(* Logix 5000 project; controller Thurs_Lab2 vendor 1 type 14 code 156 rev 30.11; software revision 30.00; part 2 of 5 *)
(* tags used below, declared in another part *)
   ALARM_CLOSE : BOOL;
   AUTO : BOOL;
   BLINK_PL1 : TIMER;
   BLINK_PL3 : TIMER;
   BLUE : BOOL;
   BLUE_BLINKER : TIMER;
   BLUE_STK : BOOL;
   BUTTON : BOOL;
   BYPASS : BOOL;
   CHECK_0 : BOOL;
   CHECK_1 : BOOL;
   CYCLE_START : BOOL;
   CYCLE_STOP : BOOL;
   CYL1_EXT_PX : BOOL;
   CYL1_RET_PX : BOOL;
   CYL2_EXT_4_LOAD_AND_UNLOAD : BOOL;
   CYL2_EXT_PX : BOOL;
   DEEP : COUNTER;
   DELAY_PE_INPUT_PSB : TIMER;
   DELAY_PE_INPUT_PSW : TIMER;
   DELAY_PE_INPUT_STATE : TIMER;
   DRILL2 : DRILL2;
   DRILL3 : DRILL3;
   DRILL4 : DRILL4;
   ESTOP : BOOL;
   ESTOP_PRESSED : BOOL;
   EXTEND : TIMER;
   FAILURE2LOAD : TIMER;
   FAILURE_2_LOAD : BOOL;
   FAULT : BOOL;
   FAULT_S : DINT;
   FAULTED : BOOL;
   FROM_CELL : FROM_CELL;
   GOOD_PART : BOOL;
   GREEN_BLINKER : TIMER;
   GREEN_STK : BOOL;
   INPUT : INT;
   LIMIT_PSB : BOOL;
   LIMIT_PSW : BOOL;
   LIMIT_STATE : BOOL;
   LOADING : BOOL;
   MACHINE_PAUSED : BOOL;
   Manual : BOOL;
   MARK_BLUE : BOOL;
   MARK_CYL1 : CYLINDER;
   MARK_GREEN : BOOL;
   MARK_LIGHTS : BOOL;
   MARK_RED : BOOL;
   MARK_WHITE_STK : BOOL;
   MARK_YELLOW : BOOL;
   MODE_SELECT : DINT;
   MOTOR_WHEEL_PE : BOOL;
   MSTER_RESET_TWCE : BOOL;
   ONESHOT1 : BOOL;
   ONESHOT2 : BOOL;
   ONESHOT3 : BOOL;
   OP1_STOP : BOOL;
   OP2_STEP : DINT;
   OP2_STOP : BOOL;
   OP2STEP : DINT;
   OP3_STOP : BOOL;
   OP4_STOP : BOOL;
   OP5_STATIC_OVER : BOOL;
   OP5_STATIC_UNDER : BOOL;
   OP5_STOP : BOOL;
   OP5_TEST : DINT;
   OP5_TEST_STATIC : DINT;
   OP6_OP7 : DINT;
   OP6_STOP : BOOL;
   OP7_STOP : BOOL;
   OPERATION : DINT;
   OPERATION_5_OVER : BOOL;
   OPERATION_5_REJECT : BOOL;
   OPERATION_5_UNDER : BOOL;
   OPERATION_7_OVER : BOOL;
   OPERATION_7_REJECT : BOOL;
   OPERATION_7_UNDER : BOOL;
   OPERATION_DONE : DINT;
   OPERATION_OFF : DINT;
   OUT_OF_INK_FAULT : BOOL;
   PART_NOT_PX : BOOL;
   PART_PX : BOOL;
   PAUSED : BOOL;
   PAUSED_OPERATION_1 : BOOL;
   PAUSED_OPERATION_5 : BOOL;
   PAUSED_OPERATION_7 : BOOL;
   PB0 : BOOL;
   PB1 : BOOL;
   PB2 : BOOL;
   PB3 : BOOL;
   PB4 : BOOL;
   PB5 : BOOL;
   PL1 : BOOL;
   PL3 : BOOL;
   PUSH : BOOL;
   PV_ANALOG_PROBE : DINT;
   PV_ANALOG_PROBE_STATIC : DINT;
   PV_CYL1_DEPTH : DINT;
   PV_CYL1_EXT_LIMIT : DINT;
   PV_CYL1_EXT_TIME : DINT;
   PV_DRILLING : DINT;
   PV_STOPPING : DINT;
   PV_UP2SPEED : DINT;
   RED_BLINKER : TIMER;
   RED_STK : BOOL;
   REJECT_FAULT : BOOL;
   RESET : BOOL;
   SAFETY_RELAY_OFF : BOOL;
   SEQ_EN : BOOL;
   SETTLE1 : TIMER;
   SHALLOW : COUNTER;
   SPARE : BOOL;
   STA : DINT;
   START_SIGNAL : BOOL;
   STATE : DINT;
   STATUS : DINT;
   STEP : DINT;
   Timer : TIMER;
   TIMER_1 : TIMER;
   TIMER_2 : TIMER;
   TO_CELL : TO_CELL;
   TOO_DEEP : BOOL;
   TOO_SHALLOW : BOOL;
   TRANSFER7 : TIMER;
   TRANSFER7_TIME_EXCEED : BOOL;
   TWO_HAND_START : BOOL;
   UNLOADING : BOOL;
   YELLOW_STK : BOOL;
(* MainProgram, continued *)

ROUTINE HMI_SCREEN   (* ladder *)
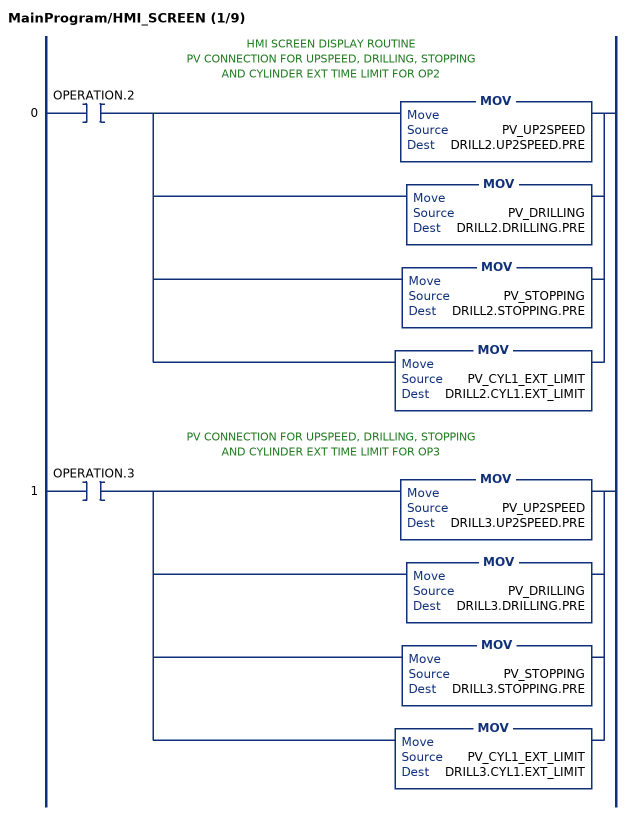
   // HMI SCREEN DISPLAY ROUTINE
   // PV CONNECTION FOR UPSPEED, DRILLING, STOPPING
   // AND CYLINDER EXT TIME LIMIT FOR OP2
   0: XIC(OPERATION.2)[MOV(PV_UP2SPEED,DRILL2.UP2SPEED.PRE) ,MOV(PV_DRILLING,DRILL2.DRILLING.PRE) ,MOV(PV_STOPPING,DRILL2.STOPPING.PRE) ,MOV(PV_CYL1_EXT_LIMIT,DRILL2.CYL1.EXT_LIMIT) ];
   // PV CONNECTION FOR UPSPEED, DRILLING, STOPPING
   // AND CYLINDER EXT TIME LIMIT FOR OP3
   1: XIC(OPERATION.3)[MOV(PV_UP2SPEED,DRILL3.UP2SPEED.PRE) ,MOV(PV_DRILLING,DRILL3.DRILLING.PRE) ,MOV(PV_STOPPING,DRILL3.STOPPING.PRE) ,MOV(PV_CYL1_EXT_LIMIT,DRILL3.CYL1.EXT_LIMIT) ];
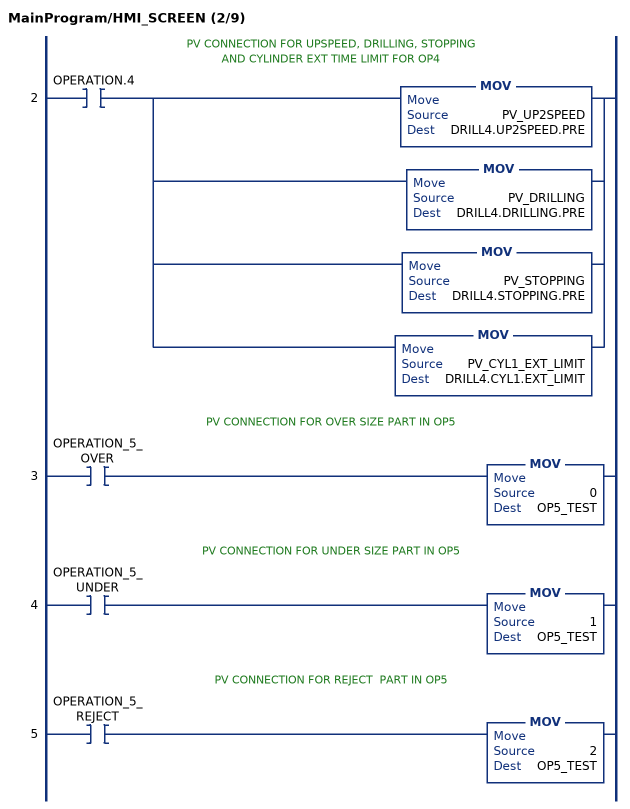
   // PV CONNECTION FOR UPSPEED, DRILLING, STOPPING
   // AND CYLINDER EXT TIME LIMIT FOR OP4
   2: XIC(OPERATION.4)[MOV(PV_UP2SPEED,DRILL4.UP2SPEED.PRE) ,MOV(PV_DRILLING,DRILL4.DRILLING.PRE) ,MOV(PV_STOPPING,DRILL4.STOPPING.PRE) ,MOV(PV_CYL1_EXT_LIMIT,DRILL4.CYL1.EXT_LIMIT) ];
   // PV CONNECTION FOR OVER SIZE PART IN OP5
   3: XIC(OPERATION_5_OVER)MOV(0,OP5_TEST);
   // PV CONNECTION FOR UNDER SIZE PART IN OP5
   4: XIC(OPERATION_5_UNDER)MOV(1,OP5_TEST);
   // PV CONNECTION FOR REJECT  PART IN OP5
   5: XIC(OPERATION_5_REJECT)MOV(2,OP5_TEST);
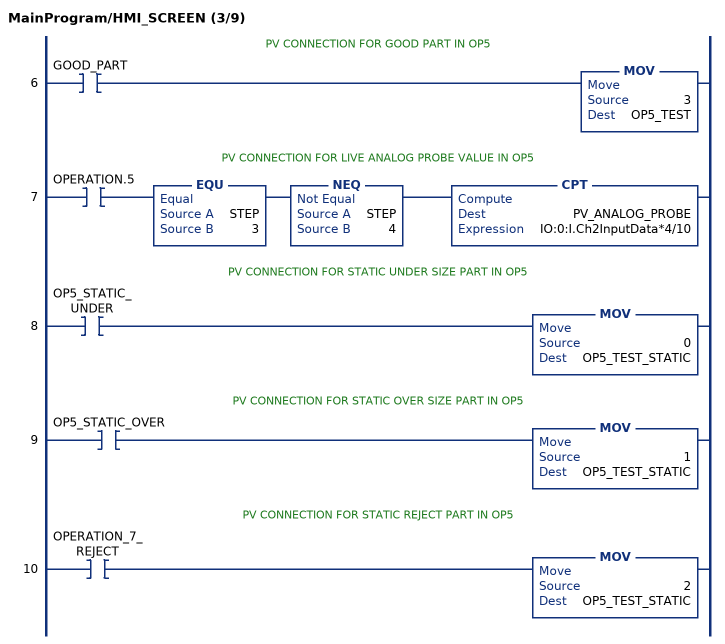
   // PV CONNECTION FOR GOOD PART IN OP5
   6: XIC(GOOD_PART)MOV(3,OP5_TEST);
   // PV CONNECTION FOR LIVE ANALOG PROBE VALUE IN OP5
   7: XIC(OPERATION.5)EQU(STEP,3)NEQ(STEP,4)CPT(PV_ANALOG_PROBE,IO:0:I.Ch2InputData*4/10);
   // PV CONNECTION FOR STATIC UNDER SIZE PART IN OP5
   8: XIC(OP5_STATIC_UNDER)MOV(0,OP5_TEST_STATIC);
   // PV CONNECTION FOR STATIC OVER SIZE PART IN OP5
   9: XIC(OP5_STATIC_OVER)MOV(1,OP5_TEST_STATIC);
   // PV CONNECTION FOR STATIC REJECT PART IN OP5
   10: XIC(OPERATION_7_REJECT)MOV(2,OP5_TEST_STATIC);
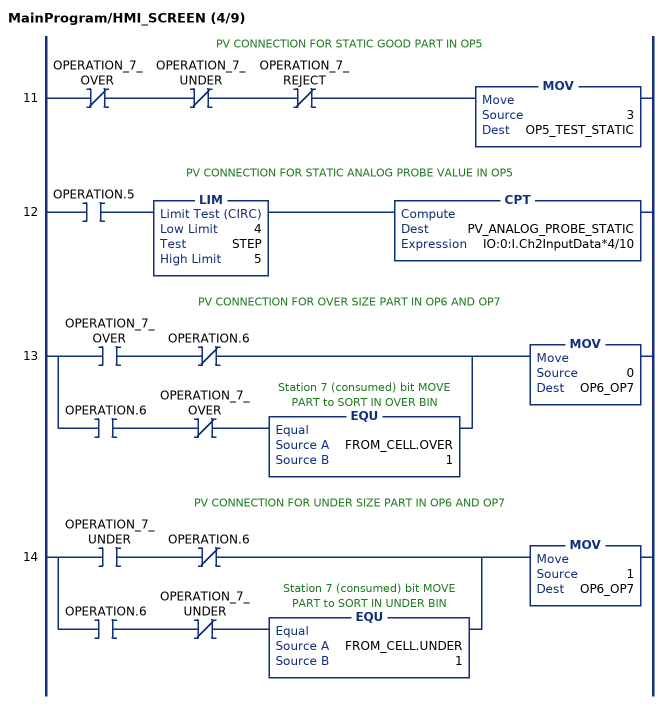
   // PV CONNECTION FOR STATIC GOOD PART IN OP5
   11: XIO(OPERATION_7_OVER)XIO(OPERATION_7_UNDER)XIO(OPERATION_7_REJECT)MOV(3,OP5_TEST_STATIC);
   // PV CONNECTION FOR STATIC ANALOG PROBE VALUE IN OP5
   12: XIC(OPERATION.5)LIM(4,STEP,5)CPT(PV_ANALOG_PROBE_STATIC,IO:0:I.Ch2InputData*4/10);
   // PV CONNECTION FOR OVER SIZE PART IN OP6 AND OP7
   13: [XIC(OPERATION_7_OVER) XIO(OPERATION.6) ,XIC(OPERATION.6) XIO(OPERATION_7_OVER) EQU(FROM_CELL.OVER,1) ]MOV(0,OP6_OP7);
   // PV CONNECTION FOR UNDER SIZE PART IN OP6 AND OP7
   14: [XIC(OPERATION_7_UNDER) XIO(OPERATION.6) ,XIC(OPERATION.6) XIO(OPERATION_7_UNDER) EQU(FROM_CELL.UNDER,1) ]MOV(1,OP6_OP7);
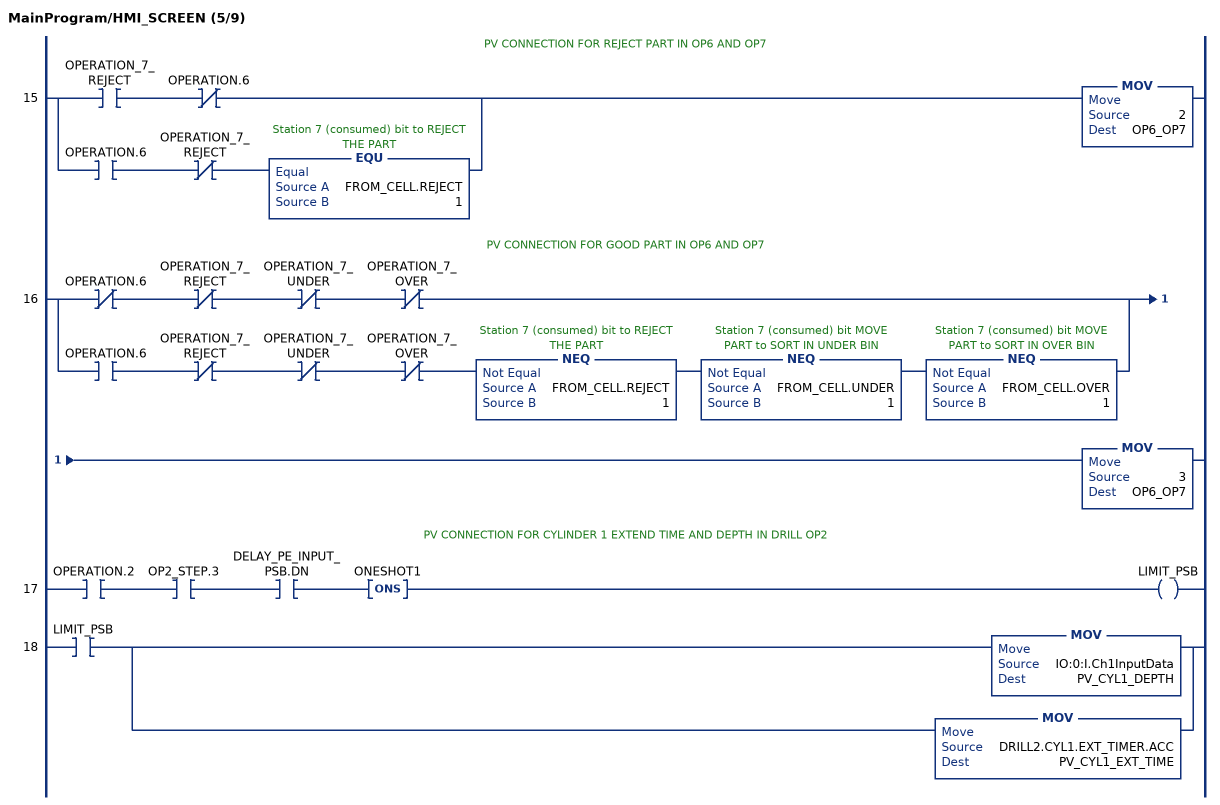
   // PV CONNECTION FOR REJECT PART IN OP6 AND OP7
   15: [XIC(OPERATION_7_REJECT) XIO(OPERATION.6) ,XIC(OPERATION.6) XIO(OPERATION_7_REJECT) EQU(FROM_CELL.REJECT,1) ]MOV(2,OP6_OP7);
   // PV CONNECTION FOR GOOD PART IN OP6 AND OP7
   16: [XIO(OPERATION.6) XIO(OPERATION_7_REJECT) XIO(OPERATION_7_UNDER) XIO(OPERATION_7_OVER) ,XIC(OPERATION.6) XIO(OPERATION_7_REJECT) XIO(OPERATION_7_UNDER) XIO(OPERATION_7_OVER) NEQ(FROM_CELL.REJECT,1) NEQ(FROM_CELL.UNDER,1) NEQ(FROM_CELL.OVER,1) ]MOV(3,OP6_OP7);
   // PV CONNECTION FOR CYLINDER 1 EXTEND TIME AND DEPTH IN DRILL OP2
   17: XIC(OPERATION.2)XIC(OP2_STEP.3)XIC(DELAY_PE_INPUT_PSB.DN)ONS(ONESHOT1)OTE(LIMIT_PSB);
   18: XIC(LIMIT_PSB)[MOV(IO:0:I.Ch1InputData,PV_CYL1_DEPTH) ,MOV(DRILL2.CYL1.EXT_TIMER.ACC,PV_CYL1_EXT_TIME) ];
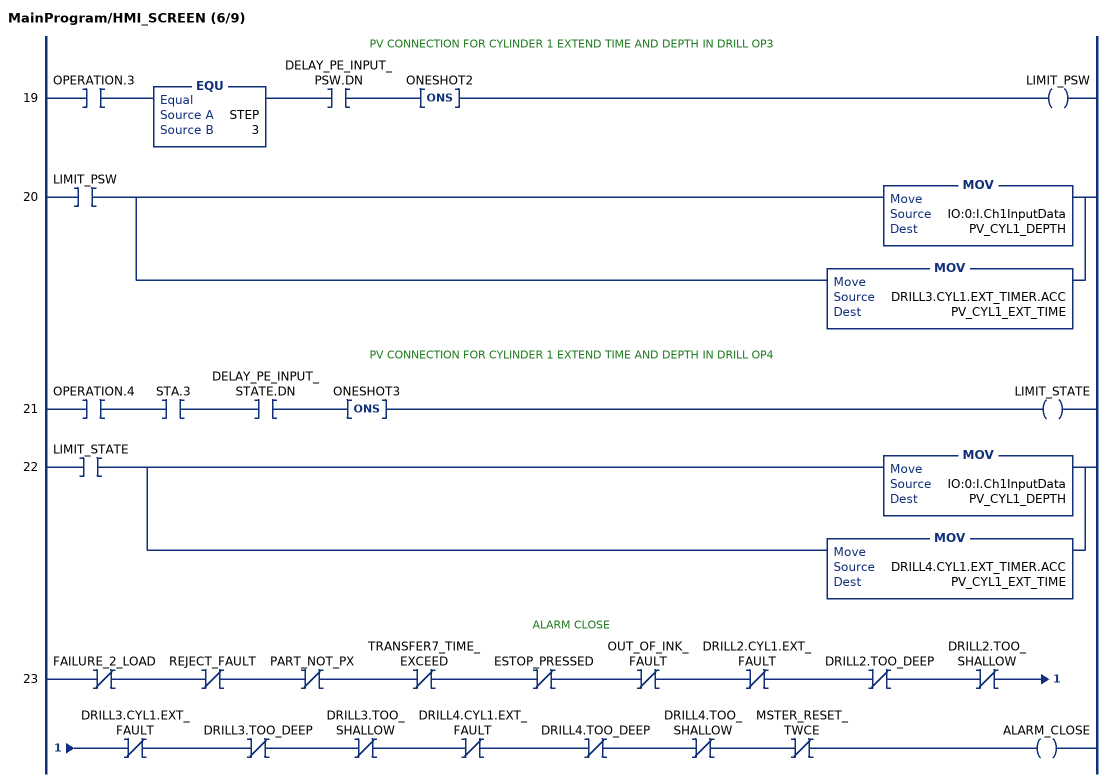
   // PV CONNECTION FOR CYLINDER 1 EXTEND TIME AND DEPTH IN DRILL OP3
   19: XIC(OPERATION.3)EQU(STEP,3)XIC(DELAY_PE_INPUT_PSW.DN)ONS(ONESHOT2)OTE(LIMIT_PSW);
   20: XIC(LIMIT_PSW)[MOV(IO:0:I.Ch1InputData,PV_CYL1_DEPTH) ,MOV(DRILL3.CYL1.EXT_TIMER.ACC,PV_CYL1_EXT_TIME) ];
   // PV CONNECTION FOR CYLINDER 1 EXTEND TIME AND DEPTH IN DRILL OP4
   21: XIC(OPERATION.4)XIC(STA.3)XIC(DELAY_PE_INPUT_STATE.DN)ONS(ONESHOT3)OTE(LIMIT_STATE);
   22: XIC(LIMIT_STATE)[MOV(IO:0:I.Ch1InputData,PV_CYL1_DEPTH) ,MOV(DRILL4.CYL1.EXT_TIMER.ACC,PV_CYL1_EXT_TIME) ];
   // ALARM CLOSE
   23: XIO(FAILURE_2_LOAD)XIO(REJECT_FAULT)XIO(PART_NOT_PX)XIO(TRANSFER7_TIME_EXCEED)XIO(ESTOP_PRESSED)XIO(OUT_OF_INK_FAULT)XIO(DRILL2.CYL1.EXT_FAULT)XIO(DRILL2.TOO_DEEP)XIO(DRILL2.TOO_SHALLOW)XIO(DRILL3.CYL1.EXT_FAULT)XIO(DRILL3.TOO_DEEP)XIO(DRILL3.TOO_SHALLOW)XIO(DRILL4.CYL1.EXT_FAULT)XIO(DRILL4.TOO_DEEP)XIO(DRILL4.TOO_SHALLOW)XIO(MSTER_RESET_TWCE)OTE(ALARM_CLOSE);
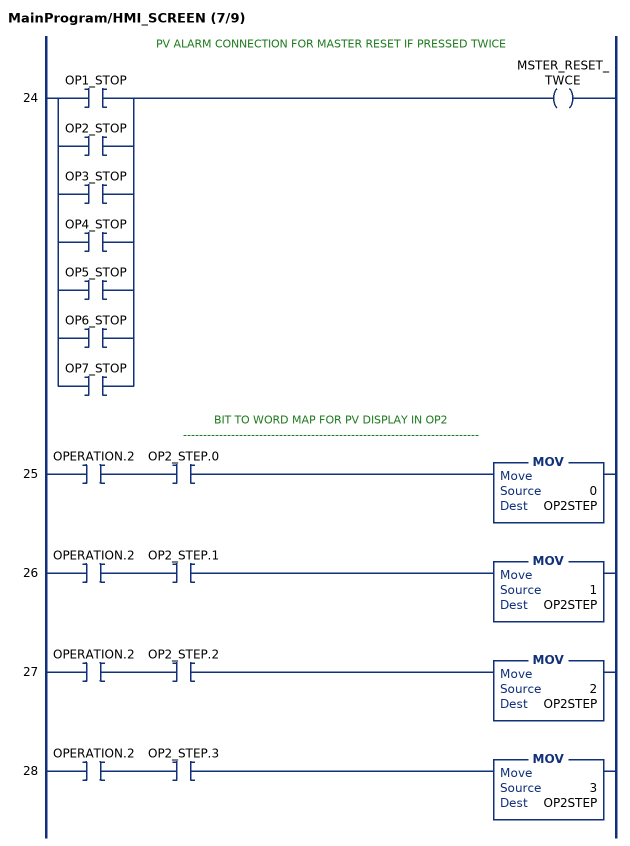
   // PV ALARM CONNECTION FOR MASTER RESET IF PRESSED TWICE
   24: [XIC(OP1_STOP) ,XIC(OP2_STOP) ,XIC(OP3_STOP) ,XIC(OP4_STOP) ,XIC(OP5_STOP) ,XIC(OP6_STOP) ,XIC(OP7_STOP) ]OTE(MSTER_RESET_TWCE);
   // BIT TO WORD MAP FOR PV DISPLAY IN OP2
   // --------------------------------------------------------------------------
   25: XIC(OPERATION.2)XIC(OP2_STEP.0)MOV(0,OP2STEP);
   26: XIC(OPERATION.2)XIC(OP2_STEP.1)MOV(1,OP2STEP);
   27: XIC(OPERATION.2)XIC(OP2_STEP.2)MOV(2,OP2STEP);
   28: XIC(OPERATION.2)XIC(OP2_STEP.3)MOV(3,OP2STEP);
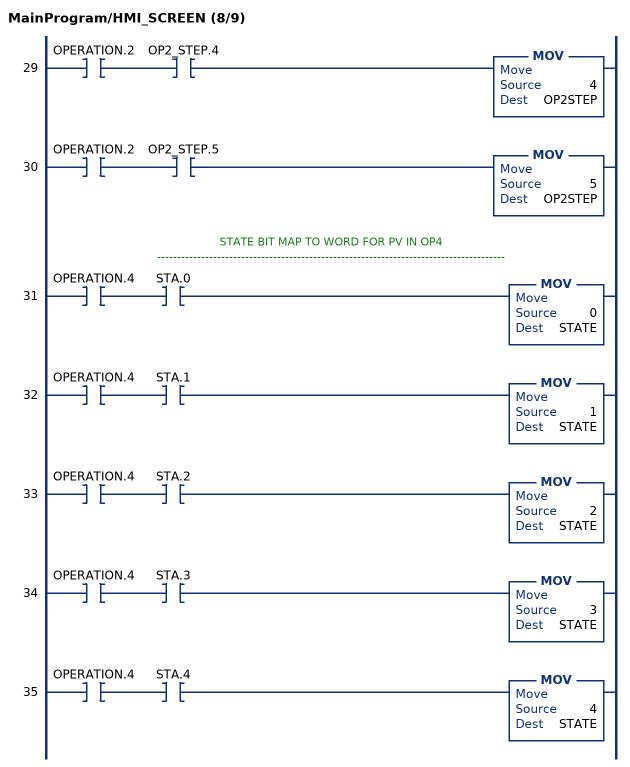
   29: XIC(OPERATION.2)XIC(OP2_STEP.4)MOV(4,OP2STEP);
   30: XIC(OPERATION.2)XIC(OP2_STEP.5)MOV(5,OP2STEP);
   // STATE BIT MAP TO WORD FOR PV IN OP4
   // ---------------------------------------------------------------------------------------
   31: XIC(OPERATION.4)XIC(STA.0)MOV(0,STATE);
   32: XIC(OPERATION.4)XIC(STA.1)MOV(1,STATE);
   33: XIC(OPERATION.4)XIC(STA.2)MOV(2,STATE);
   34: XIC(OPERATION.4)XIC(STA.3)MOV(3,STATE);
   35: XIC(OPERATION.4)XIC(STA.4)MOV(4,STATE);
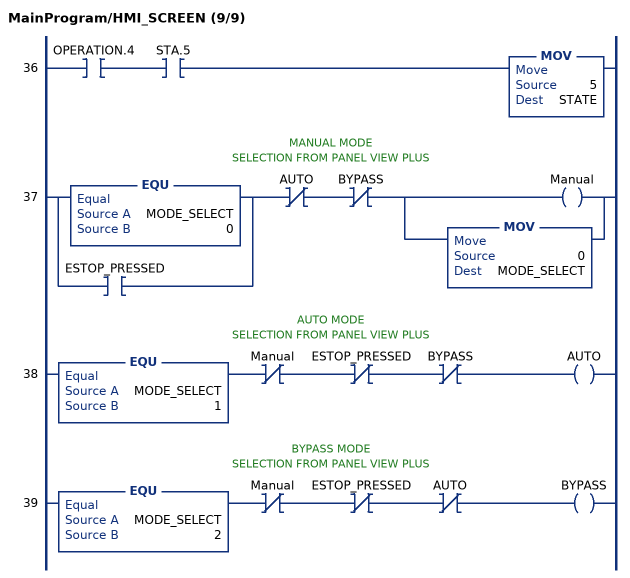
   36: XIC(OPERATION.4)XIC(STA.5)MOV(5,STATE);
   // MANUAL MODE
   // SELECTION FROM PANEL VIEW PLUS
   37: [EQU(MODE_SELECT,0) ,XIC(ESTOP_PRESSED) ]XIO(AUTO)XIO(BYPASS)[OTE(Manual) ,MOV(0,MODE_SELECT) ];
   // AUTO MODE
   // SELECTION FROM PANEL VIEW PLUS
   38: EQU(MODE_SELECT,1)XIO(Manual)XIO(ESTOP_PRESSED)XIO(BYPASS)OTE(AUTO);
   // BYPASS MODE
   // SELECTION FROM PANEL VIEW PLUS
   39: EQU(MODE_SELECT,2)XIO(Manual)XIO(ESTOP_PRESSED)XIO(AUTO)OTE(BYPASS);
END_ROUTINE

ROUTINE INDICATOR   (* ladder *)
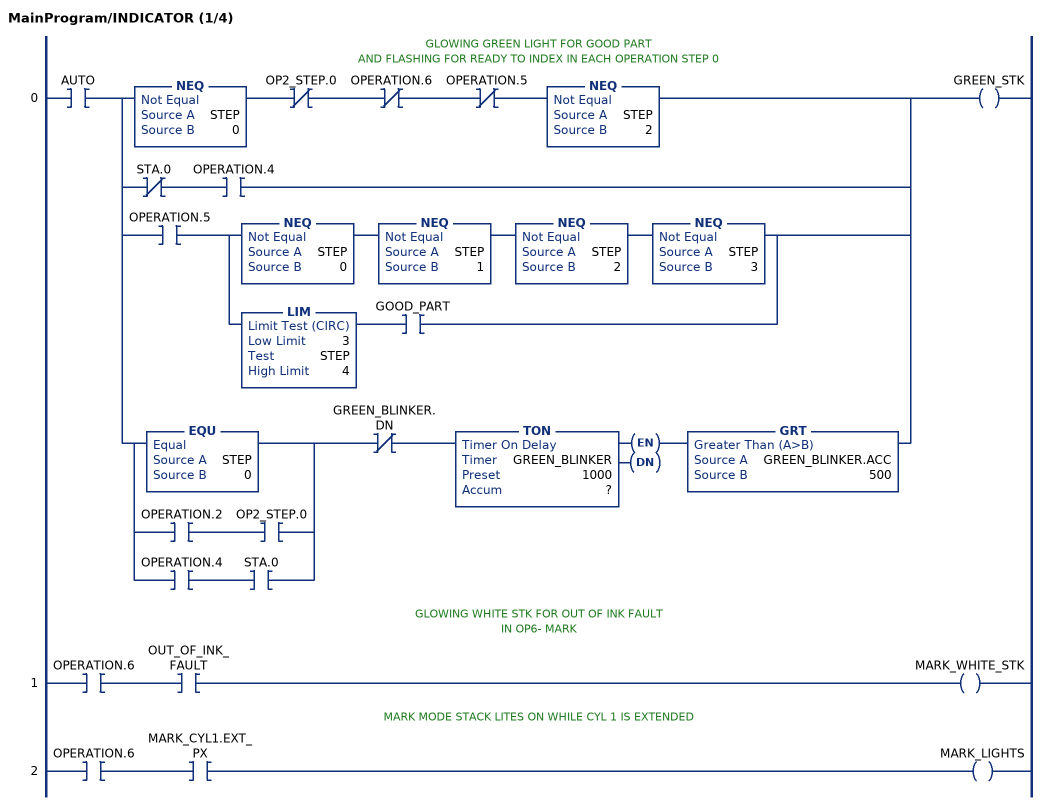
   // GLOWING GREEN LIGHT FOR GOOD PART
   // AND FLASHING FOR READY TO INDEX IN EACH OPERATION STEP 0
   0: XIC(AUTO)[[[NEQ(STEP,0) XIO(OP2_STEP.0) XIO(OPERATION.6) XIO(OPERATION.5) NEQ(STEP,2) ,XIO(STA.0) XIC(OPERATION.4) ] ,XIC(OPERATION.5) [NEQ(STEP,0) NEQ(STEP,1) NEQ(STEP,2) NEQ(STEP,3) ,LIM(3,STEP,4) XIC(GOOD_PART) ] ] ,[EQU(STEP,0) ,XIC(OPERATION.2) XIC(OP2_STEP.0) ,XIC(OPERATION.4) XIC(STA.0) ] XIO(GREEN_BLINKER.DN) TON(GREEN_BLINKER,?,?) GRT(GREEN_BLINKER.ACC,500) ]OTE(GREEN_STK);
   // GLOWING WHITE STK FOR OUT OF INK FAULT
   // IN OP6- MARK
   1: XIC(OPERATION.6)XIC(OUT_OF_INK_FAULT)OTE(MARK_WHITE_STK);
   // MARK MODE STACK LITES ON WHILE CYL 1 IS EXTENDED
   2: XIC(OPERATION.6)XIC(MARK_CYL1.EXT_PX)OTE(MARK_LIGHTS);
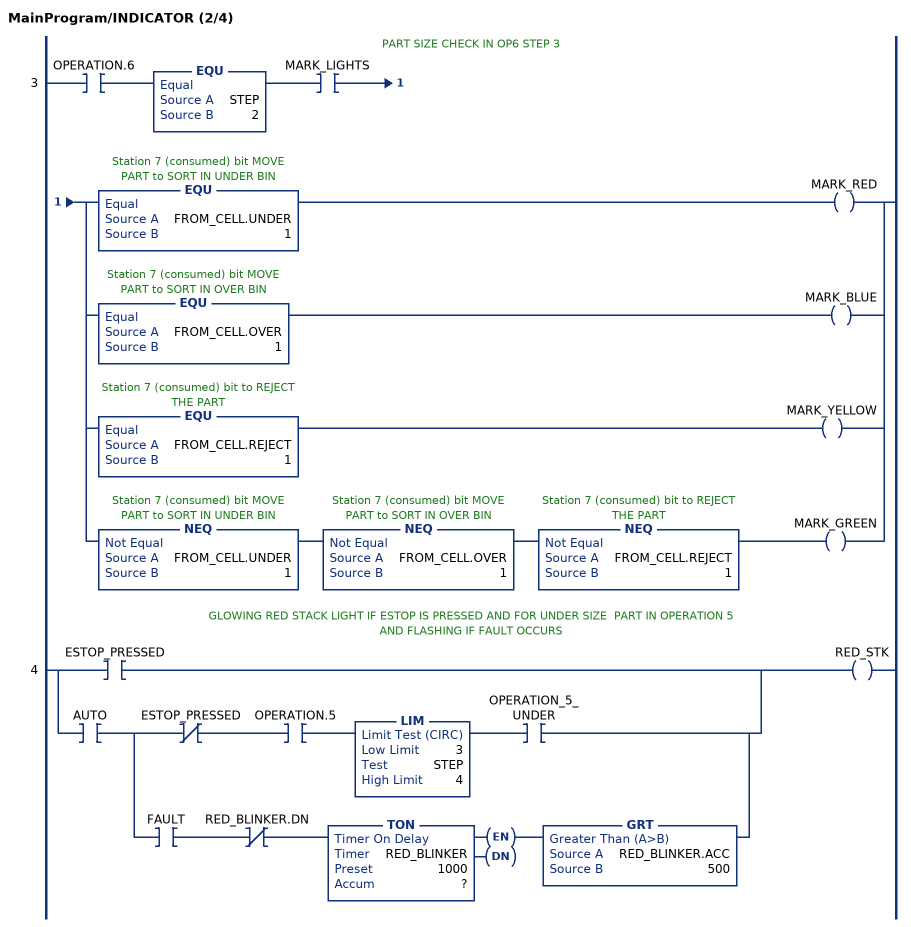
   // PART SIZE CHECK IN OP6 STEP 3
   3: XIC(OPERATION.6)EQU(STEP,2)XIC(MARK_LIGHTS)[EQU(FROM_CELL.UNDER,1) OTE(MARK_RED) ,EQU(FROM_CELL.OVER,1) OTE(MARK_BLUE) ,EQU(FROM_CELL.REJECT,1) OTE(MARK_YELLOW) ,NEQ(FROM_CELL.UNDER,1) NEQ(FROM_CELL.OVER,1) NEQ(FROM_CELL.REJECT,1) OTE(MARK_GREEN) ];
   // GLOWING RED STACK LIGHT IF ESTOP IS PRESSED AND FOR UNDER SIZE  PART IN OPERATION 5
   // AND FLASHING IF FAULT OCCURS
   4: [XIC(ESTOP_PRESSED) ,XIC(AUTO) [XIO(ESTOP_PRESSED) XIC(OPERATION.5) LIM(3,STEP,4) XIC(OPERATION_5_UNDER) ,XIC(FAULT) XIO(RED_BLINKER.DN) TON(RED_BLINKER,?,?) GRT(RED_BLINKER.ACC,500) ] ]OTE(RED_STK);
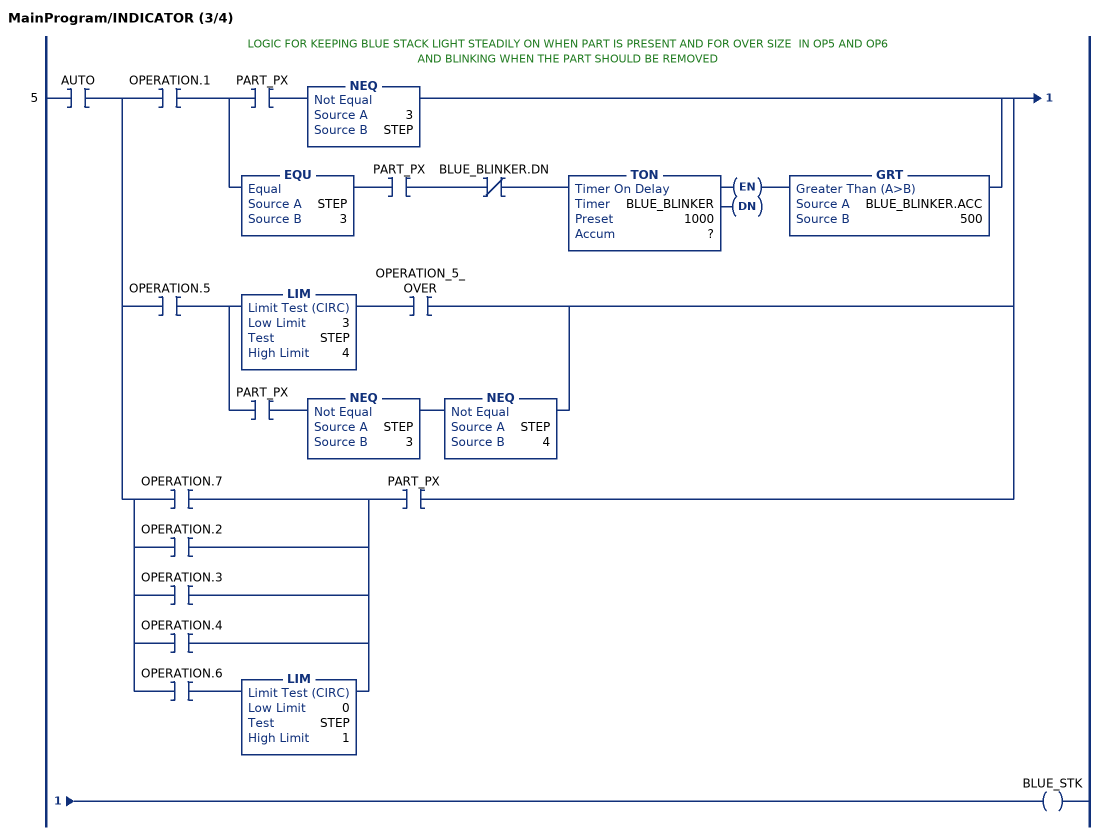
   // LOGIC FOR KEEPING BLUE STACK LIGHT STEADILY ON WHEN PART IS PRESENT AND FOR OVER SIZE  IN OP5 AND OP6
   // AND BLINKING WHEN THE PART SHOULD BE REMOVED
   5: XIC(AUTO)[XIC(OPERATION.1) [XIC(PART_PX) NEQ(3,STEP) ,EQU(STEP,3) XIC(PART_PX) XIO(BLUE_BLINKER.DN) TON(BLUE_BLINKER,?,?) GRT(BLUE_BLINKER.ACC,500) ] ,XIC(OPERATION.5) [LIM(3,STEP,4) XIC(OPERATION_5_OVER) ,XIC(PART_PX) NEQ(STEP,3) NEQ(STEP,4) ] ,[XIC(OPERATION.7) ,XIC(OPERATION.2) ,XIC(OPERATION.3) ,XIC(OPERATION.4) ,XIC(OPERATION.6) LIM(0,STEP,1) ] XIC(PART_PX) ]OTE(BLUE_STK);
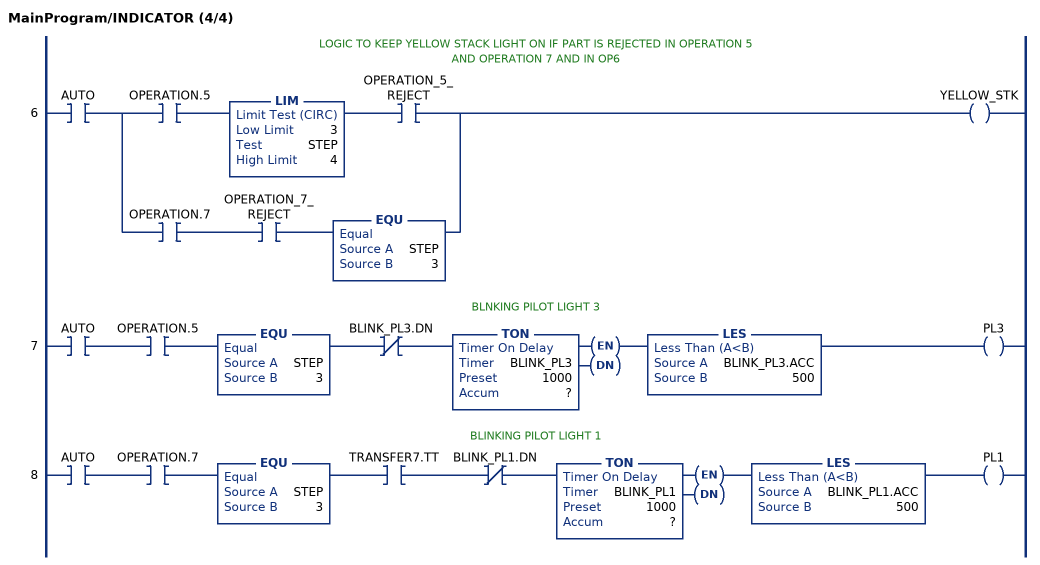
   // LOGIC TO KEEP YELLOW STACK LIGHT ON IF PART IS REJECTED IN OPERATION 5
   // AND OPERATION 7 AND IN OP6
   6: XIC(AUTO)[XIC(OPERATION.5) LIM(3,STEP,4) XIC(OPERATION_5_REJECT) ,XIC(OPERATION.7) XIC(OPERATION_7_REJECT) EQU(STEP,3) ]OTE(YELLOW_STK);
   // BLNKING PILOT LIGHT 3
   7: XIC(AUTO)XIC(OPERATION.5)EQU(STEP,3)XIO(BLINK_PL3.DN)TON(BLINK_PL3,?,?)LES(BLINK_PL3.ACC,500)OTE(PL3);
   // BLINKING PILOT LIGHT 1
   8: XIC(AUTO)XIC(OPERATION.7)EQU(STEP,3)XIC(TRANSFER7.TT)XIO(BLINK_PL1.DN)TON(BLINK_PL1,?,?)LES(BLINK_PL1.ACC,500)OTE(PL1);
END_ROUTINE

ROUTINE INPUT_BUFFERING   (* structured text *)
   // STRUCTURED TEXT PROGRAMMING FOR INPUT BUFFERING ROUTINE
   
   PB0 := Local:1:I.Data.0; // BUFFERING FOR PUSH BUTTON 0
   PB1 := Local:1:I.Data.1; //	BUFFERING FOR PUSH BUTTON 1
   PB2 := Local:1:I.Data.2; //	BUFFERING FOR PUSH BUTTON 2
   PB3 := Local:1:I.Data.3; //	BUFFERING FOR PUSH BUTTON 3
   PB4 := Local:1:I.Data.4; //	BUFFERING FOR PUSH BUTTON 4
   PB5 := Local:1:I.Data.5; //	BUFFERING FOR PUSH BUTTON 5
   
   CYL2_EXT_PX := Local:1:I.Data.6; //	BUFFERING FOR CYLINDER 2 EXTEND PROX
   MOTOR_WHEEL_PE:= Local:1:I.Data.7;	//	BUFFERING FOR MOTOR WHEEL PHOTO EYE
   PART_PX := Local:1:I.Data.8 AND (NOT PB2); //	BUFFERING FOR PART PRESENT AND INTERLOCKED WITH PB2
   SPARE:= Local:1:I.Data.9;
   
   CYL1_EXT_PX := Local:1:I.Data.10; //	BUFFERING CYLINDER 1 EXT PROX
   DRILL2.CYL1.EXT_PX := Local:1:I.Data.10;
   DRILL3.CYL1.EXT_PX := Local:1:I.Data.10;
   DRILL4.CYL1.EXT_PX := Local:1:I.Data.10;
   MARK_CYL1.EXT_PX := Local:1:I.Data.10;
   
   CYL1_RET_PX := Local:1:I.Data.11; //	BUFFERING FOR CYLINDER 1 EXTEND PROX
   DRILL2.CYL1.RET_PX := Local:1:I.Data.11;
   DRILL3.CYL1.RET_PX:= Local:1:I.Data.11;
   DRILL4.CYL1.RET_PX := Local:1:I.Data.11;
   MARK_CYL1.RET_PX := Local:1:I.Data.11;
   
   CYCLE_STOP := Local:1:I.Data.12;	//	BUFFERING FOR CYCLE STOP
   CYCLE_START := Local:1:I.Data.13;	//	BUFFERING FOR CYCLE START
   ESTOP_PRESSED := Local:1:I.Data.14;  //	BUFFERING FOR ESTOP PRESS
   SAFETY_RELAY_OFF:= Local:1:I.Data.15; // BUFFERING FOR SAFETY RELAY
   
   
   
END_ROUTINE

ROUTINE LOAD_UNLOADING   (* ladder *)
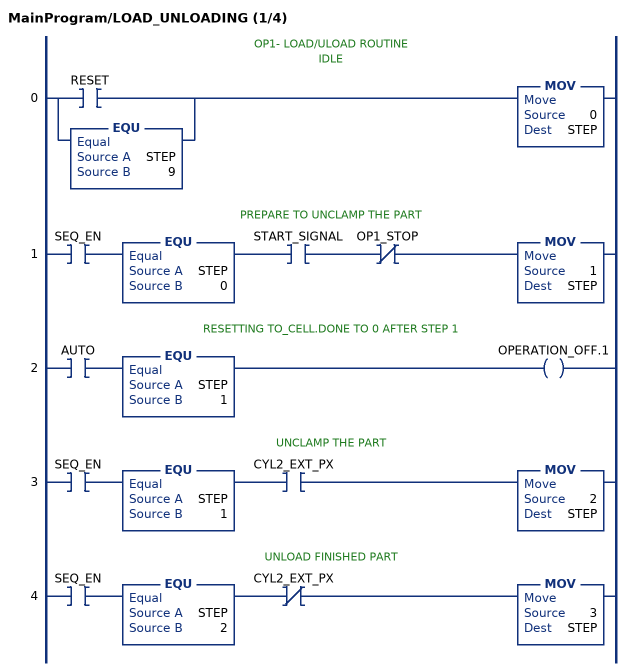
   // OP1- LOAD/ULOAD ROUTINE
   // IDLE
   0: [XIC(RESET) ,EQU(STEP,9) ]MOV(0,STEP);
   // PREPARE TO UNCLAMP THE PART
   1: XIC(SEQ_EN)EQU(STEP,0)XIC(START_SIGNAL)XIO(OP1_STOP)MOV(1,STEP);
   // RESETTING TO_CELL.DONE TO 0 AFTER STEP 1
   2: XIC(AUTO)EQU(STEP,1)OTE(OPERATION_OFF.1);
   // UNCLAMP THE PART
   3: XIC(SEQ_EN)EQU(STEP,1)XIC(CYL2_EXT_PX)MOV(2,STEP);
   // UNLOAD FINISHED PART
   4: XIC(SEQ_EN)EQU(STEP,2)XIO(CYL2_EXT_PX)MOV(3,STEP);
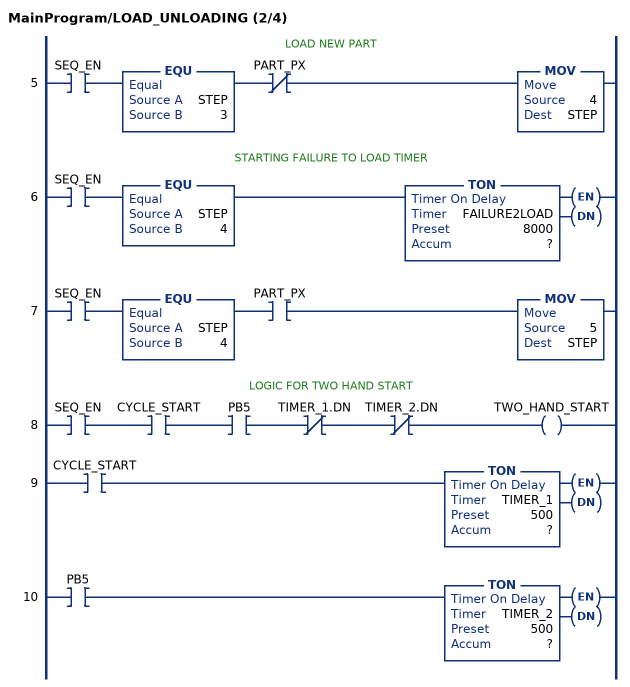
   // LOAD NEW PART
   5: XIC(SEQ_EN)EQU(STEP,3)XIO(PART_PX)MOV(4,STEP);
   // STARTING FAILURE TO LOAD TIMER
   6: XIC(SEQ_EN)EQU(STEP,4)TON(FAILURE2LOAD,?,?);
   7: XIC(SEQ_EN)EQU(STEP,4)XIC(PART_PX)MOV(5,STEP);
   // LOGIC FOR TWO HAND START
   8: XIC(SEQ_EN)XIC(CYCLE_START)XIC(PB5)XIO(TIMER_1.DN)XIO(TIMER_2.DN)OTE(TWO_HAND_START);
   9: XIC(CYCLE_START)TON(TIMER_1,?,?);
   10: XIC(PB5)TON(TIMER_2,?,?);
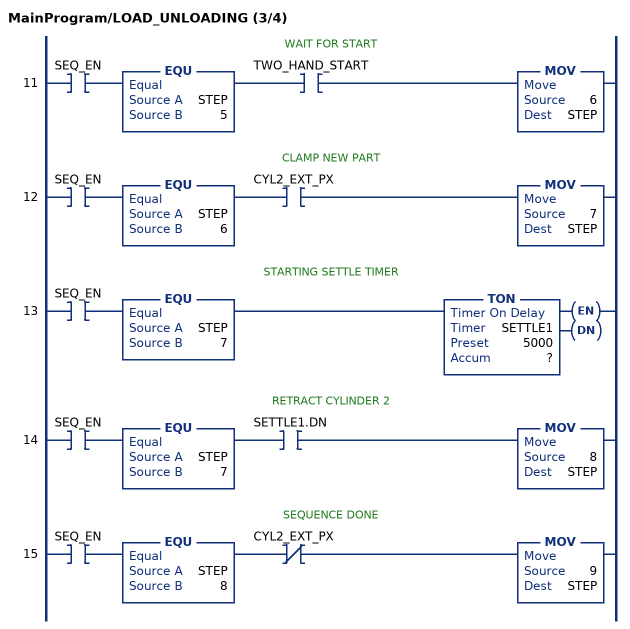
   // WAIT FOR START
   11: XIC(SEQ_EN)EQU(STEP,5)XIC(TWO_HAND_START)MOV(6,STEP);
   // CLAMP NEW PART
   12: XIC(SEQ_EN)EQU(STEP,6)XIC(CYL2_EXT_PX)MOV(7,STEP);
   // STARTING SETTLE TIMER
   13: XIC(SEQ_EN)EQU(STEP,7)TON(SETTLE1,?,?);
   // RETRACT CYLINDER 2
   14: XIC(SEQ_EN)EQU(STEP,7)XIC(SETTLE1.DN)MOV(8,STEP);
   // SEQUENCE DONE
   15: XIC(SEQ_EN)EQU(STEP,8)XIO(CYL2_EXT_PX)MOV(9,STEP);
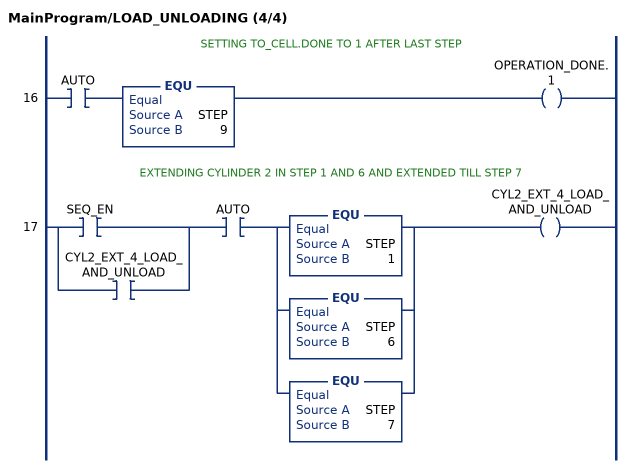
   // SETTING TO_CELL.DONE TO 1 AFTER LAST STEP
   16: XIC(AUTO)EQU(STEP,9)OTE(OPERATION_DONE.1);
   // EXTENDING CYLINDER 2 IN STEP 1 AND 6 AND EXTENDED TILL STEP 7
   17: [XIC(SEQ_EN) ,XIC(CYL2_EXT_4_LOAD_AND_UNLOAD) ]XIC(AUTO)[EQU(STEP,1) ,EQU(STEP,6) ,EQU(STEP,7) ]OTE(CYL2_EXT_4_LOAD_AND_UNLOAD);
END_ROUTINE

ROUTINE MACHINE_STATUS_AND_FAULTS   (* ladder *)
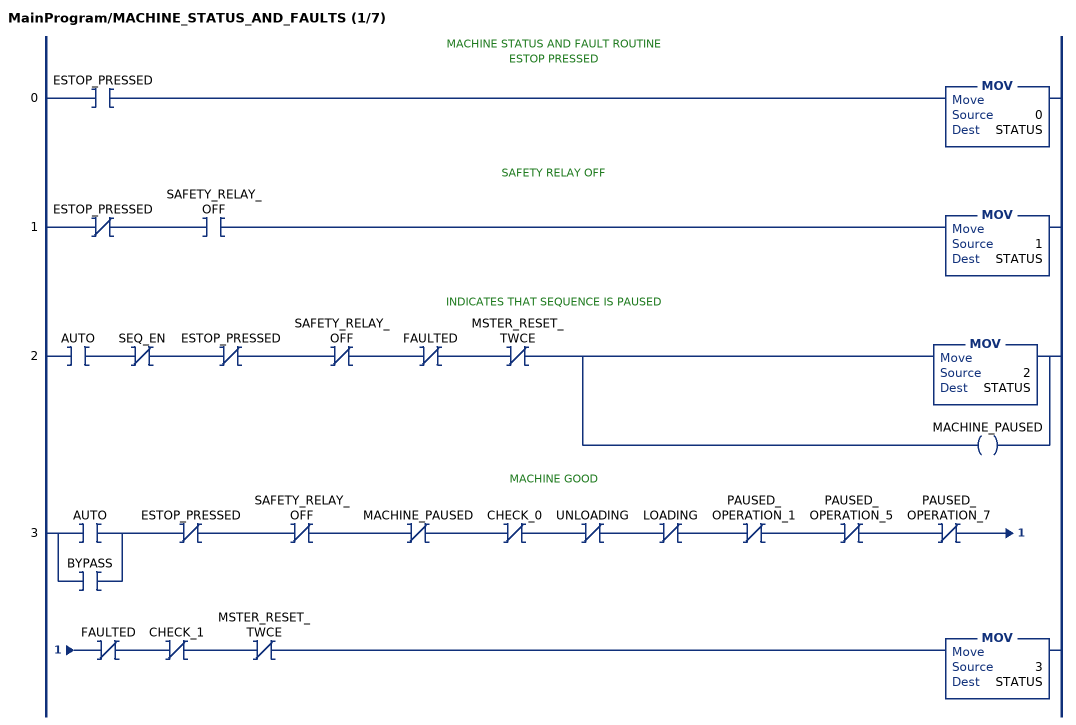
   // MACHINE STATUS AND FAULT ROUTINE
   // ESTOP PRESSED
   0: XIC(ESTOP_PRESSED)MOV(0,STATUS);
   // SAFETY RELAY OFF
   1: XIO(ESTOP_PRESSED)XIC(SAFETY_RELAY_OFF)MOV(1,STATUS);
   // INDICATES THAT SEQUENCE IS PAUSED
   2: XIC(AUTO)XIO(SEQ_EN)XIO(ESTOP_PRESSED)XIO(SAFETY_RELAY_OFF)XIO(FAULTED)XIO(MSTER_RESET_TWCE)[MOV(2,STATUS) ,OTE(MACHINE_PAUSED) ];
   // MACHINE GOOD
   3: [XIC(AUTO) ,XIC(BYPASS) ]XIO(ESTOP_PRESSED)XIO(SAFETY_RELAY_OFF)XIO(MACHINE_PAUSED)XIO(CHECK_0)XIO(UNLOADING)XIO(LOADING)XIO(PAUSED_OPERATION_1)XIO(PAUSED_OPERATION_5)XIO(PAUSED_OPERATION_7)XIO(FAULTED)XIO(CHECK_1)XIO(MSTER_RESET_TWCE)MOV(3,STATUS);
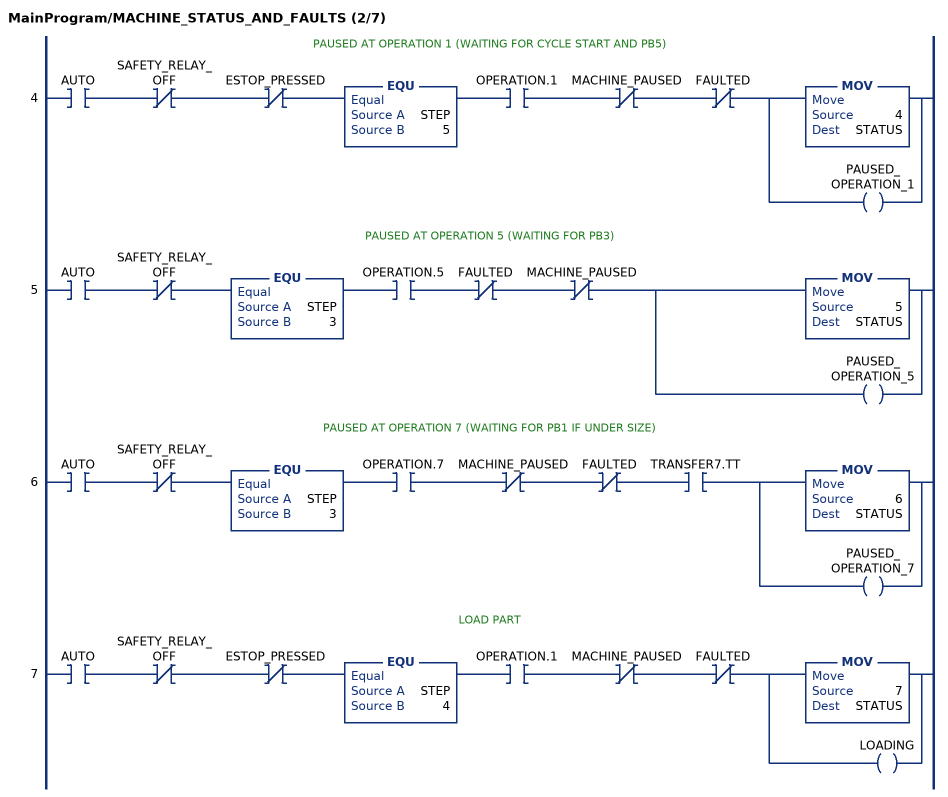
   // PAUSED AT OPERATION 1 (WAITING FOR CYCLE START AND PB5)
   4: XIC(AUTO)XIO(SAFETY_RELAY_OFF)XIO(ESTOP_PRESSED)EQU(STEP,5)XIC(OPERATION.1)XIO(MACHINE_PAUSED)XIO(FAULTED)[MOV(4,STATUS) ,OTE(PAUSED_OPERATION_1) ];
   // PAUSED AT OPERATION 5 (WAITING FOR PB3)
   5: XIC(AUTO)XIO(SAFETY_RELAY_OFF)EQU(STEP,3)XIC(OPERATION.5)XIO(FAULTED)XIO(MACHINE_PAUSED)[MOV(5,STATUS) ,OTE(PAUSED_OPERATION_5) ];
   // PAUSED AT OPERATION 7 (WAITING FOR PB1 IF UNDER SIZE)
   6: XIC(AUTO)XIO(SAFETY_RELAY_OFF)EQU(STEP,3)XIC(OPERATION.7)XIO(MACHINE_PAUSED)XIO(FAULTED)XIC(TRANSFER7.TT)[MOV(6,STATUS) ,OTE(PAUSED_OPERATION_7) ];
   // LOAD PART
   7: XIC(AUTO)XIO(SAFETY_RELAY_OFF)XIO(ESTOP_PRESSED)EQU(STEP,4)XIC(OPERATION.1)XIO(MACHINE_PAUSED)XIO(FAULTED)[MOV(7,STATUS) ,OTE(LOADING) ];
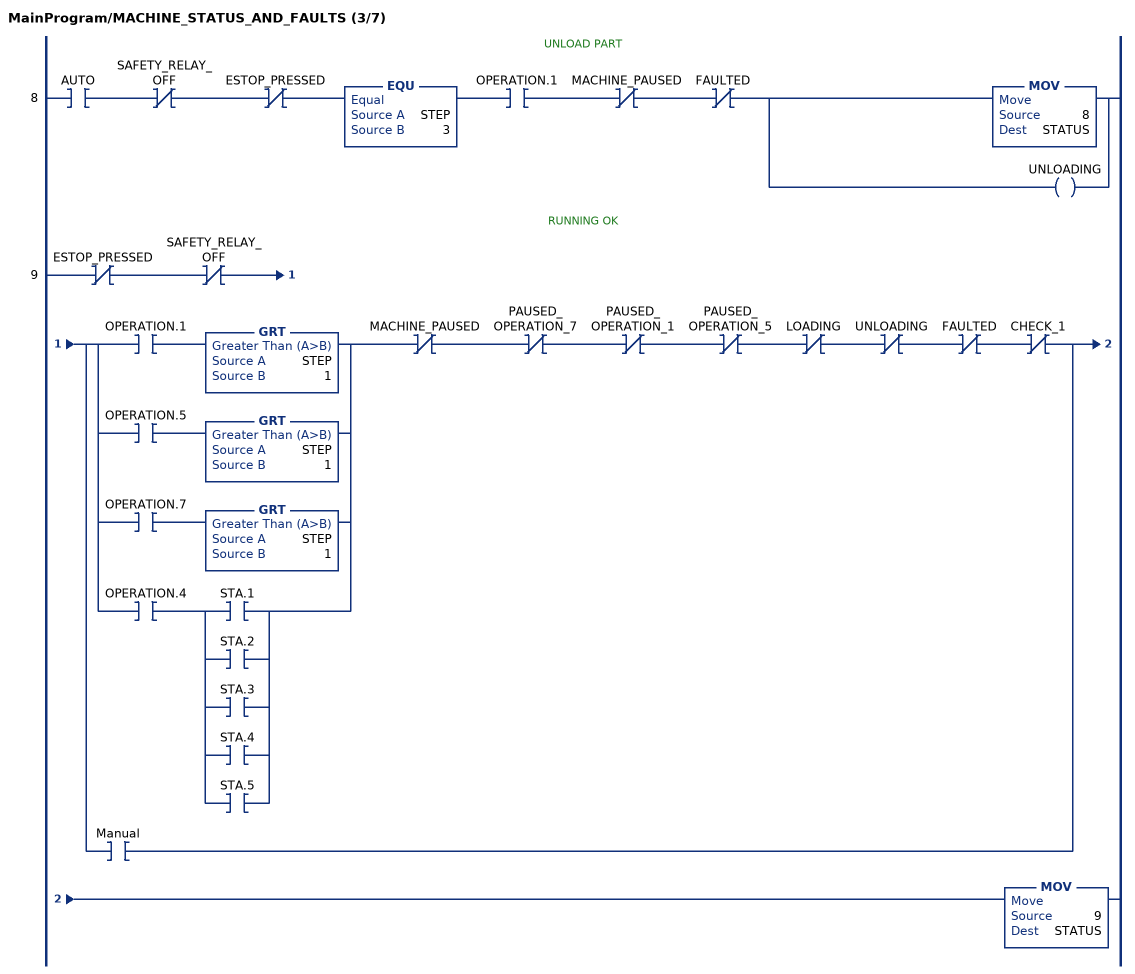
   // UNLOAD PART
   8: XIC(AUTO)XIO(SAFETY_RELAY_OFF)XIO(ESTOP_PRESSED)EQU(STEP,3)XIC(OPERATION.1)XIO(MACHINE_PAUSED)XIO(FAULTED)[MOV(8,STATUS) ,OTE(UNLOADING) ];
   // RUNNING OK
   9: XIO(ESTOP_PRESSED)XIO(SAFETY_RELAY_OFF)[[XIC(OPERATION.1) GRT(STEP,1) ,XIC(OPERATION.5) GRT(STEP,1) ,XIC(OPERATION.7) GRT(STEP,1) ,XIC(OPERATION.4) [XIC(STA.1) ,XIC(STA.2) ,XIC(STA.3) ,XIC(STA.4) ,XIC(STA.5) ] ] XIO(MACHINE_PAUSED) XIO(PAUSED_OPERATION_7) XIO(PAUSED_OPERATION_1) XIO(PAUSED_OPERATION_5) XIO(LOADING) XIO(UNLOADING) XIO(FAULTED) XIO(CHECK_1) ,XIC(Manual) ]MOV(9,STATUS);
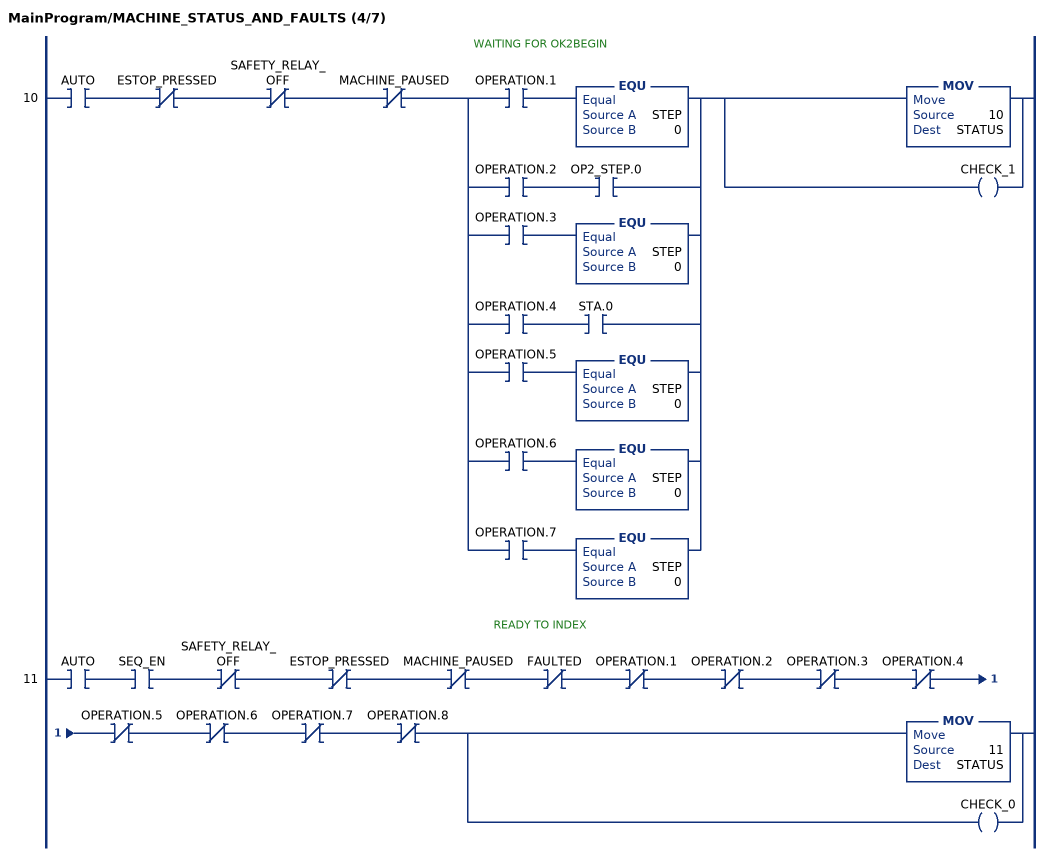
   // WAITING FOR OK2BEGIN
   10: XIC(AUTO)XIO(ESTOP_PRESSED)XIO(SAFETY_RELAY_OFF)XIO(MACHINE_PAUSED)[XIC(OPERATION.1) EQU(STEP,0) ,XIC(OPERATION.2) XIC(OP2_STEP.0) ,XIC(OPERATION.3) EQU(STEP,0) ,XIC(OPERATION.4) XIC(STA.0) ,XIC(OPERATION.5) EQU(STEP,0) ,XIC(OPERATION.6) EQU(STEP,0) ,XIC(OPERATION.7) EQU(STEP,0) ][MOV(10,STATUS) ,OTE(CHECK_1) ];
   // READY TO INDEX
   11: XIC(AUTO)XIC(SEQ_EN)XIO(SAFETY_RELAY_OFF)XIO(ESTOP_PRESSED)XIO(MACHINE_PAUSED)XIO(FAULTED)XIO(OPERATION.1)XIO(OPERATION.2)XIO(OPERATION.3)XIO(OPERATION.4)XIO(OPERATION.5)XIO(OPERATION.6)XIO(OPERATION.7)XIO(OPERATION.8)[MOV(11,STATUS) ,OTE(CHECK_0) ];
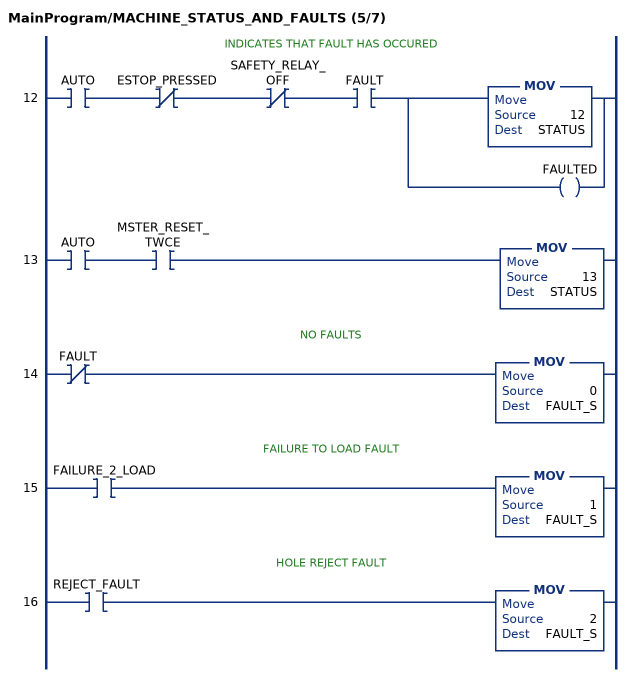
   // INDICATES THAT FAULT HAS OCCURED
   12: XIC(AUTO)XIO(ESTOP_PRESSED)XIO(SAFETY_RELAY_OFF)XIC(FAULT)[MOV(12,STATUS) ,OTE(FAULTED) ];
   13: XIC(AUTO)XIC(MSTER_RESET_TWCE)MOV(13,STATUS);
   // NO FAULTS
   14: XIO(FAULT)MOV(0,FAULT_S);
   // FAILURE TO LOAD FAULT
   15: XIC(FAILURE_2_LOAD)MOV(1,FAULT_S);
   // HOLE REJECT FAULT
   16: XIC(REJECT_FAULT)MOV(2,FAULT_S);
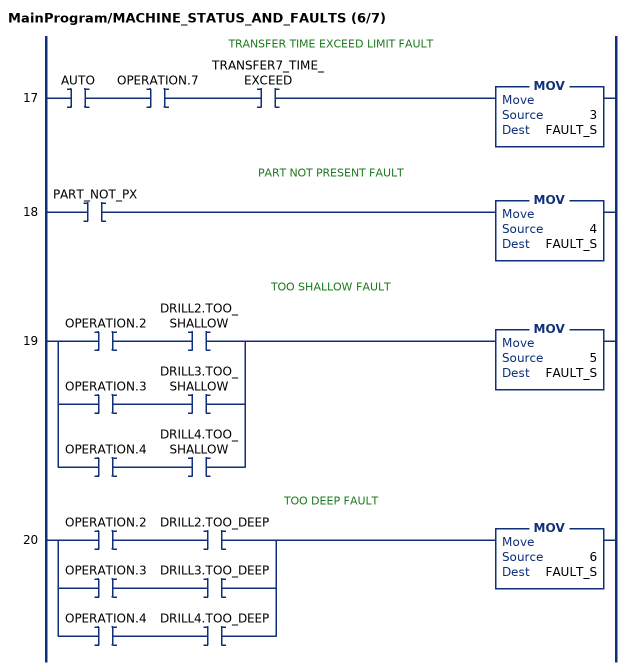
   // TRANSFER TIME EXCEED LIMIT FAULT
   17: XIC(AUTO)XIC(OPERATION.7)XIC(TRANSFER7_TIME_EXCEED)MOV(3,FAULT_S);
   // PART NOT PRESENT FAULT
   18: XIC(PART_NOT_PX)MOV(4,FAULT_S);
   // TOO SHALLOW FAULT
   19: [XIC(OPERATION.2) XIC(DRILL2.TOO_SHALLOW) ,XIC(OPERATION.3) XIC(DRILL3.TOO_SHALLOW) ,XIC(OPERATION.4) XIC(DRILL4.TOO_SHALLOW) ]MOV(5,FAULT_S);
   // TOO DEEP FAULT
   20: [XIC(OPERATION.2) XIC(DRILL2.TOO_DEEP) ,XIC(OPERATION.3) XIC(DRILL3.TOO_DEEP) ,XIC(OPERATION.4) XIC(DRILL4.TOO_DEEP) ]MOV(6,FAULT_S);
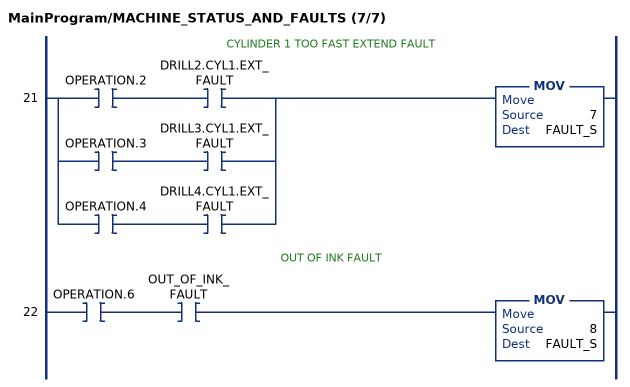
   // CYLINDER 1 TOO FAST EXTEND FAULT
   21: [XIC(OPERATION.2) XIC(DRILL2.CYL1.EXT_FAULT) ,XIC(OPERATION.3) XIC(DRILL3.CYL1.EXT_FAULT) ,XIC(OPERATION.4) XIC(DRILL4.CYL1.EXT_FAULT) ]MOV(7,FAULT_S);
   // OUT OF INK FAULT
   22: XIC(OPERATION.6)XIC(OUT_OF_INK_FAULT)MOV(8,FAULT_S);
END_ROUTINE
